FUNCTION_BLOCK FB_InfluxMessage
VAR_INPUT
	// payload string received
	sPayload:	STRING(255);
END_VAR
VAR_OUTPUT
	// measurement string (first word)
	measurement:	STRING(255) := '';
	// parameter (variable name)
	parameter:		STRING(255) := '';
	// value (variable content)
	value:			STRING(255) := '';
	// the payload for the NEXT parameter=value pair ("measurement[,tags] rest-of-field-set[ timestamp]"),
	// '' if this was the last pair. Feed it back in as sPayload to walk a multi-field message.
	remaining:		STRING(255) := '';
END_VAR
VAR
	space_position:		INT;
	//equial_position:	INT;
	comma_position:		INT;
	measurement_tags:	STRING(255);
	parameter_value: 	STRING(255);
	bResultSplit: 		BOOL;
	sRest:				STRING(255);
	// definition of the space separator
	spaceSeparator:		STRING(1) := ' ';
	// definition of the comma separator
	commaSeparator:		STRING(1) := ',';
	// definition of the equial sign separator
	equialSeparator:	STRING(1) := '=';
END_VAR

(* 
parse message in influx format:
	measurement parameter=value
	measurement,tag1=tag1value parameter=value
	measurement,tag1=tag1value parameter1=value1,parameter2=value2 [timestamp]

Returns the FIRST parameter=value pair. If there are more, 'remaining' holds a complete payload for the next
pair (measurement and tags in front, timestamp kept at the end), so the caller feeds it straight back in.
Tags are accepted but not returned. A quoted string value that contains a comma or a space is not handled.
*)

// start from empty outputs every call: a caller that reuses the instance must not see the previous pair again
measurement := '';
parameter := '';
value := '';
remaining := '';

//separate measurement from parameter, value
bResultSplit := FindAndSplit( pSeparator     := ADR(spaceSeparator), pSrcString := ADR(sPayload), 
                              pLeftString    := ADR(measurement_tags), nLeftSize  := SIZEOF(measurement_tags), 
                              pRightString   := ADR(parameter_value), nRightSize := SIZEOF(parameter_value),
                              bSearchFromRight := FALSE );
IF NOT bResultSplit THEN
	RETURN;
END_IF
// look for tags attached to the measurement
comma_position := FIND(measurement_tags, commaSeparator);
IF comma_position = 0 THEN
	measurement := measurement_tags;
ELSE
	measurement := LEFT(measurement_tags, comma_position-1);
END_IF
// dissect the parameter=value part
comma_position := FIND(parameter_value, commaSeparator);
IF comma_position = 0 THEN
	// we have only one parameter value pair
	bResultSplit := FindAndSplit( pSeparator     := ADR(equialSeparator), pSrcString := ADR(parameter_value), 
                              pLeftString    := ADR(parameter), nLeftSize  := SIZEOF(parameter), 
                              pRightString   := ADR(value), nRightSize := SIZEOF(value),
                              bSearchFromRight := FALSE );

ELSE
	// we have more than one parameter value pair: everything after the first comma is the next pair(s),
	// handed back with the measurement and tags in front (the space between them was consumed above)
	sRest := MID(parameter_value, LEN(parameter_value) - comma_position, comma_position + 1);
	remaining := CONCAT(CONCAT(measurement_tags, spaceSeparator), sRest);
	parameter_value := LEFT(parameter_value, comma_position-1);
	bResultSplit := FindAndSplit( pSeparator     := ADR(equialSeparator), pSrcString := ADR(parameter_value), 
                              pLeftString    := ADR(parameter), nLeftSize  := SIZEOF(parameter), 
                              pRightString   := ADR(value), nRightSize := SIZEOF(value),
                              bSearchFromRight := FALSE );
END_IF

// a trailing Influx timestamp (measurement[,tags] field_set timestamp) ends up appended to value,
// since only the first space in the whole payload is split off above; drop it and anything after
// the first remaining space. A genuine quoted string value could itself contain a space, but this
// parser doesn't handle that either way (see the module comment's TODOs)
space_position := FIND(value, spaceSeparator);
IF space_position > 0 THEN
	value := LEFT(value, space_position-1);
END_IF

// strip the surrounding quotes Influx line protocol uses for a string-typed field value
IF LEN(value) >= 2 AND LEFT(value,1) = '"' AND RIGHT(value,1) = '"' THEN
	value := MID(value, LEN(value)-2, 2);
END_IF

END_FUNCTION_BLOCK

(* stored: Version 1.1.0.1, ProductVersion 3.1.4024.12
   POU FB_InfluxMessage: Id {90ca1cc6-8109-4bcf-9f8e-c5cf65cdb4b2}, SpecialFunc None *)
